// TIA Portal project "2022.06.02_电机正反转" (V17)

(* hardware
DEVICE "S7-1200 station_1"  S7-1200 Station
   slot 0: "Rack_0"  S7-1200 Rack  Rack  V1.0
   slot 1: "PLC_1"  CPU 1212C DC/DC/DC  6ES7 212-1AE40-0XB0  V4.5
*)

// ===== PLC "PLC_1"  CPU 1212C DC/DC/DC =====

VAR_GLOBAL   // PLC tag table "默认变量表"
   "System_Byte" AT %MB1 : Byte;
   "FirstScan" AT %M1.0 : Bool;
   "DiagStatusUpdate" AT %M1.1 : Bool;
   "AlwaysTRUE" AT %M1.2 : Bool;
   "AlwaysFALSE" AT %M1.3 : Bool;
   "Clock_Byte" AT %MB0 : Byte;
   "Clock_10Hz" AT %M0.0 : Bool;
   "Clock_5Hz" AT %M0.1 : Bool;
   "Clock_2.5Hz" AT %M0.2 : Bool;
   "Clock_2Hz" AT %M0.3 : Bool;
   "Clock_1.25Hz" AT %M0.4 : Bool;
   "Clock_1Hz" AT %M0.5 : Bool;
   "Clock_0.625Hz" AT %M0.6 : Bool;
   "Clock_0.5Hz" AT %M0.7 : Bool;
   "正启动" AT %I0.1 : Bool;
   "停止" AT %I0.3 : Bool;
   "反转" AT %Q0.1 : Bool;
   "正转" AT %Q0.0 : Bool;
   "反启动" AT %I0.2 : Bool;
END_VAR

ORGANIZATION_BLOCK "Main"   // OB1, LAD, ProgramCycle
TITLE = "Main Program Sweep (Cycle)"
{ S7_Optimized_Access := 'TRUE' }
VERSION : 0.1
   VAR_INPUT
      Initial_Call : Bool;   // Initial call of this OB
      Remanence : Bool;   // =True, if remanent data are available
   END_VAR
BEGIN

REGION Network 1
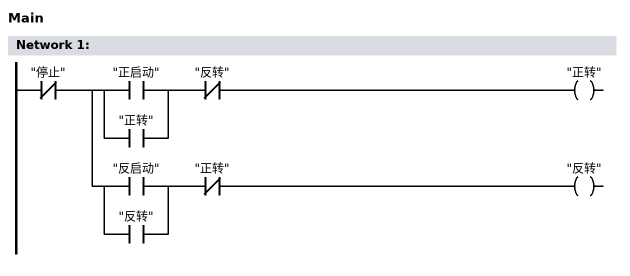
   RUNG wire#powerrail
      I_Contact( "停止" )
      wire#w1
      Contact( "正启动" )
      wire#w2
      I_Contact( "反转" )
      Coil( "正转" )
   END_RUNG
   RUNG wire#w1
      Contact( "正转" )
   END_RUNG wire#w2
   RUNG wire#w1
      Contact( "反启动" )
      wire#w3
      I_Contact( "正转" )
      Coil( "反转" )
   END_RUNG
   RUNG wire#w1
      Contact( "反转" )
   END_RUNG wire#w3
   // the same network as SCL:
   "正转" := NOT "停止" AND ("正启动" OR "正转") AND NOT "反转";
   "反转" := NOT "停止" AND ("反启动" OR "反转") AND NOT "正转";
END_REGION
END_ORGANIZATION_BLOCK